// TIA Portal V20 export
FUNCTION_BLOCK "FB_PusherControl"   // FB3, LAD
TITLE = Pusher Control
// Pusher ram sequencing (C-118-C-125). Step legend (C-120): 0=Idle (no motion; home is the HomeLimit switch, not implied by the step - after a jog release the ram may legitimately rest off home, REQ-039) - 10=DriveToEndTravel (forward stroke in progress) - 20=Hold (paused at full travel, brief settle before retracting) - 30=Retract (returning to home; also the recovery/abort target from any bad state). Mode legend: 0=Off (finish a retract already in progress, then park; no new cycle starts) - 1=Auto (hopper-high-level starts a cycle) - 2=Manual (operator button/jog starts a cycle). Motion policy (owner rulings 2026-07-16): an idle off-home ram reparks ONLY on the plant pre-start ParkCmd or on a live cycle request - never on jog release or bare mode changes - and every motion start from rest (repark, cycle launch, jog) is preceded by the JogWarningTime sounder warning (NEW-4: no unwarned pusher motion). CycleInhibit (any live plant stop reason) blocks cycle launches and aborts an in-flight cycle to park, but deliberately leaves hand-jog available - only the mode-0 force (stop button/unhealthy) blocks jogging (owner amendment 2026-07-16, REQ-040). Fitted=FALSE (REQ-042/043/044) kills every demand, the pack output, both supervision timers, and every fault latch at the source, so a disabled pusher does nothing and raises nothing. A live drop mid-cycle also force-parks Step to 0/Idle rather than stranding it non-zero (owner ruling 2026-07-17, B-4, NETWORK 14) - re-enabling Fitted is never itself a start condition (C-128): the normal Step 0 launch/repark gates (NETWORK 1) still require a fresh live trigger before anything moves again.
   VAR RETAIN
      IO { S7_SetPoint := 'True'} : "UDT_PusherIO";   // Caller-visible interface (C-115) - FC_ControlMain writes Mode/HopperHighLevel/limits/tunables in, reads Extend/Retract/RunPowerPack/fault bits out. See the block header for the Step/Mode value legend.
   END_VAR
   VAR
      CycleRequest : Bool;   // Named once, read everywhere (C-601): the live cycle trigger - Auto on hopper high or Manual on the HMI button - gated by Enable (Fitted AND not Off) and NOT Blocked. Read by the warning armer, the launch and repark transitions, and the trip-count reset. Blocked is written later in the scan, so this reads it one scan behind - immaterial: Blocked can only latch mid-stroke (Step 10) where no Step 0 request can act, and a reset-clear merely delays a relaunch by one scan.
      JogDemand : Bool;   // A live jog request: either jog button held, idle, Manual mode, pusher fitted. Arms the pre-motion warning, suppresses the repark (jogging is never fought by an auto-retract), and - per direction, warning done - drives the demands. Reads Step from before this scan's transitions; the demand rungs re-check Step fresh.
      ReparkRequest : Bool;   // A repark to home is wanted: the sequencer's pre-start ParkCmd (REQ-045) or a live CycleRequest, while idle off home and not jogging. One of the only two motion sources out of Step 0 (owner ruling 2026-07-16); fires the 0-to-30 transition once the pre-motion warning has sounded.
      LaunchRequest : Bool;   // A cycle launch is possible: live CycleRequest, idle, ram at home. Fires the 0-to-10 transition once the pre-motion warning has sounded; the same fired condition resets PressureTripCount (per-cycle jam counting, REQ-048).
      CycleAbort : Bool;   // Named once (C-601): abort an in-flight cycle to Retract - Off commanded mid-cycle, or the plant acquired a stop reason (CycleInhibit). Read by the Step 10 and Step 20 exits; the Step 30 retract completes regardless, so an aborted cycle always ends parked. Jog is untouched by this bit (owner amendment 2026-07-16).
      EndTravelTimeoutMS : DInt;
      ParkedTimeoutMS : DInt;
      EndTravelHoldTimeMS : DInt;
      PumpRunOnTimeMS : DInt;
      JogWarningTimeMS : DInt;
      PressureTripConfirmTimeMS : DInt;
      PressureClearResumeDelayMS : DInt;
      PressureConfirmTimer { S7_SetPoint := 'True'} : TON_TIME;
      PressureClearTimer { S7_SetPoint := 'True'} : TON_TIME;
      PressureHold : Bool;   // Latched jam hold, not a fault (C-123) - see the Pressure Detection network. Freezes ExtendDemand while set; clears itself once pressure has genuinely stayed clear for PressureClearResumeDelay.
      PressureConfirmEdge : Bool;
      PressureConfirmEdgeMem : Bool;
      PressureTripCount : Int;   // Confirmed jams this cycle - reset each cycle start, not time-windowed. Compared against IO.PressureTripCountThreshold to raise Blocked.
      EndTravelTimer { S7_SetPoint := 'True'} : TON_TIME;
      HoldTimer { S7_SetPoint := 'True'} : TON_TIME;
      ParkedTimer { S7_SetPoint := 'True'} : TON_TIME;
      JogPreStartTimer { S7_SetPoint := 'True'} : TON_TIME;
      ExtendDemand : Bool;
      RetractDemand : Bool;
      PumpDemand : Bool;   // ExtendDemand OR RetractDemand - the pump's own immediate (non-run-on) demand signal.
      PumpEverDemanded : Bool;   // Cold-start guard for the pump run-on off-delay below - see that network's own comment.
      PumpRunOnTimer { S7_SetPoint := 'True'} : TON_TIME;
   END_VAR
   VAR_TEMP
      "Time" : Real;
   END_VAR
BEGIN

REGION Network 1: Enable And Motion Requests
   // The compound conditions every later network shares, each written once (C-601). Requests read Step as it settled last scan (the transitions run later) - safe, because Step only ever leaves 0 through this scan's own request-gated transitions; steps returning to 0 just re-arm the requests one scan late. CycleInhibit kills cycle requests (no launch into a stopped plant) and, via CycleAbort, retracts an in-flight cycle - while JogDemand deliberately ignores it: hand-jog stays available with the plant stopped by downstream absence (owner amendment 2026-07-16, REQ-040).
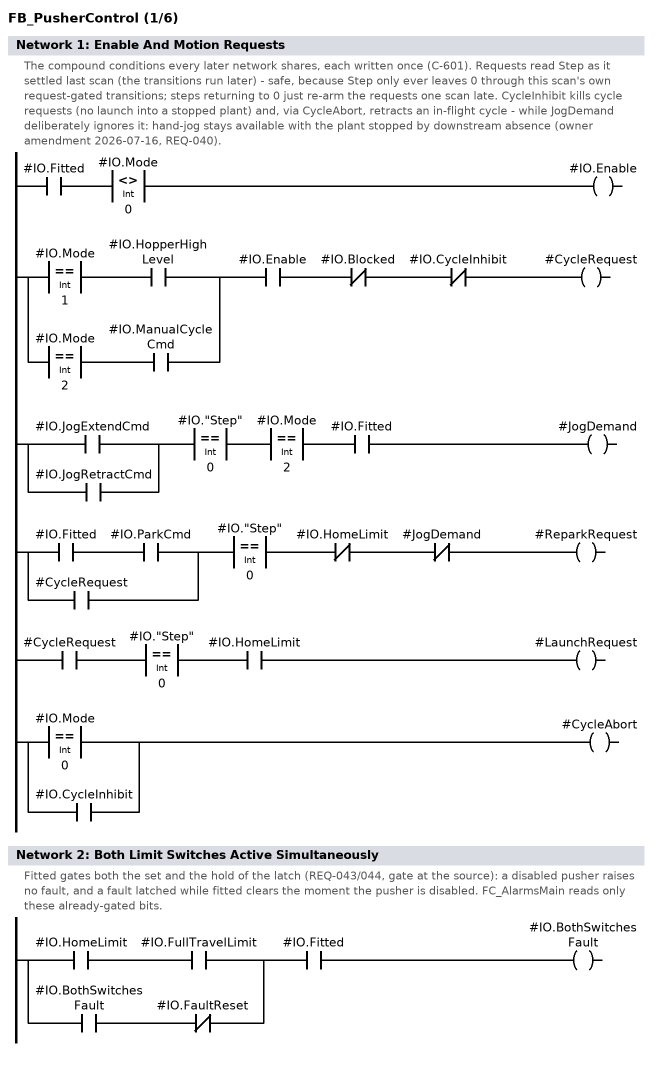
   RUNG wire#powerrail
      Contact( #IO.Fitted )
      { S7_Templates := "SrcType := Int" } NE_Contact(in1 := #IO.Mode, in2 := 0)
      Coil( #IO.Enable )
   END_RUNG
   RUNG wire#powerrail
      { S7_Templates := "SrcType := Int" } EQ_Contact(in1 := #IO.Mode, in2 := 1)
      Contact( #IO.HopperHighLevel )
      wire#w1
      Contact( #IO.Enable )
      I_Contact( #IO.Blocked )
      I_Contact( #IO.CycleInhibit )
      Coil( #CycleRequest )
   END_RUNG
   RUNG wire#powerrail
      { S7_Templates := "SrcType := Int" } EQ_Contact(in1 := #IO.Mode, in2 := 2)
      Contact( #IO.ManualCycleCmd )
   END_RUNG wire#w1
   RUNG wire#powerrail
      Contact( #IO.JogExtendCmd )
      wire#w2
      { S7_Templates := "SrcType := Int" } EQ_Contact(in1 := #IO."Step", in2 := 0)
      { S7_Templates := "SrcType := Int" } EQ_Contact(in1 := #IO.Mode, in2 := 2)
      Contact( #IO.Fitted )
      Coil( #JogDemand )
   END_RUNG
   RUNG wire#powerrail
      Contact( #IO.JogRetractCmd )
   END_RUNG wire#w2
   RUNG wire#powerrail
      Contact( #IO.Fitted )
      Contact( #IO.ParkCmd )
      wire#w3
      { S7_Templates := "SrcType := Int" } EQ_Contact(in1 := #IO."Step", in2 := 0)
      I_Contact( #IO.HomeLimit )
      I_Contact( #JogDemand )
      Coil( #ReparkRequest )
   END_RUNG
   RUNG wire#powerrail
      Contact( #CycleRequest )
   END_RUNG wire#w3
   RUNG wire#powerrail
      Contact( #CycleRequest )
      { S7_Templates := "SrcType := Int" } EQ_Contact(in1 := #IO."Step", in2 := 0)
      Contact( #IO.HomeLimit )
      Coil( #LaunchRequest )
   END_RUNG
   RUNG wire#powerrail
      { S7_Templates := "SrcType := Int" } EQ_Contact(in1 := #IO.Mode, in2 := 0)
      wire#w4
      Coil( #CycleAbort )
   END_RUNG
   RUNG wire#powerrail
      Contact( #IO.CycleInhibit )
   END_RUNG wire#w4
   // the same network as SCL:
   #IO.Enable := #IO.Fitted AND (#IO.Mode <> 0);
   #CycleRequest := (((#IO.Mode = 1) AND #IO.HopperHighLevel) OR ((#IO.Mode = 2) AND #IO.ManualCycleCmd)) AND #IO.Enable AND NOT #IO.Blocked AND NOT #IO.CycleInhibit;
   #JogDemand := (#IO.JogExtendCmd OR #IO.JogRetractCmd) AND (#IO."Step" = 0) AND (#IO.Mode = 2) AND #IO.Fitted;
   #ReparkRequest := ((#IO.Fitted AND #IO.ParkCmd) OR #CycleRequest) AND (#IO."Step" = 0) AND NOT #IO.HomeLimit AND NOT #JogDemand;
   #LaunchRequest := #CycleRequest AND (#IO."Step" = 0) AND #IO.HomeLimit;
   #CycleAbort := (#IO.Mode = 0) OR #IO.CycleInhibit;
END_REGION

REGION Network 2: Both Limit Switches Active Simultaneously
   // Fitted gates both the set and the hold of the latch (REQ-043/044, gate at the source): a disabled pusher raises no fault, and a fault latched while fitted clears the moment the pusher is disabled. FC_AlarmsMain reads only these already-gated bits.
   RUNG wire#powerrail
      Contact( #IO.HomeLimit )
      Contact( #IO.FullTravelLimit )
      wire#w1
      Contact( #IO.Fitted )
      Coil( #IO.BothSwitchesFault )
   END_RUNG
   RUNG wire#powerrail
      Contact( #IO.BothSwitchesFault )
      I_Contact( #IO.FaultReset )
   END_RUNG wire#w1
   // the same network as SCL:
   #IO.BothSwitchesFault := ((#IO.HomeLimit AND #IO.FullTravelLimit) OR (#IO.BothSwitchesFault AND NOT #IO.FaultReset)) AND #IO.Fitted;
END_REGION

REGION Network 3: HMI Time Conversions
   // HMI/DB_Settings times are Real seconds for operator legibility; every TON below needs its PT in DInt ms - one MUL+CONVERT pair per timer, matching the MotorDOL FTTime/EnableUPSTime idiom. Kept as one block up front rather than repeated at each timer, so the x1000 idiom is visibly consistent and only ever done once.
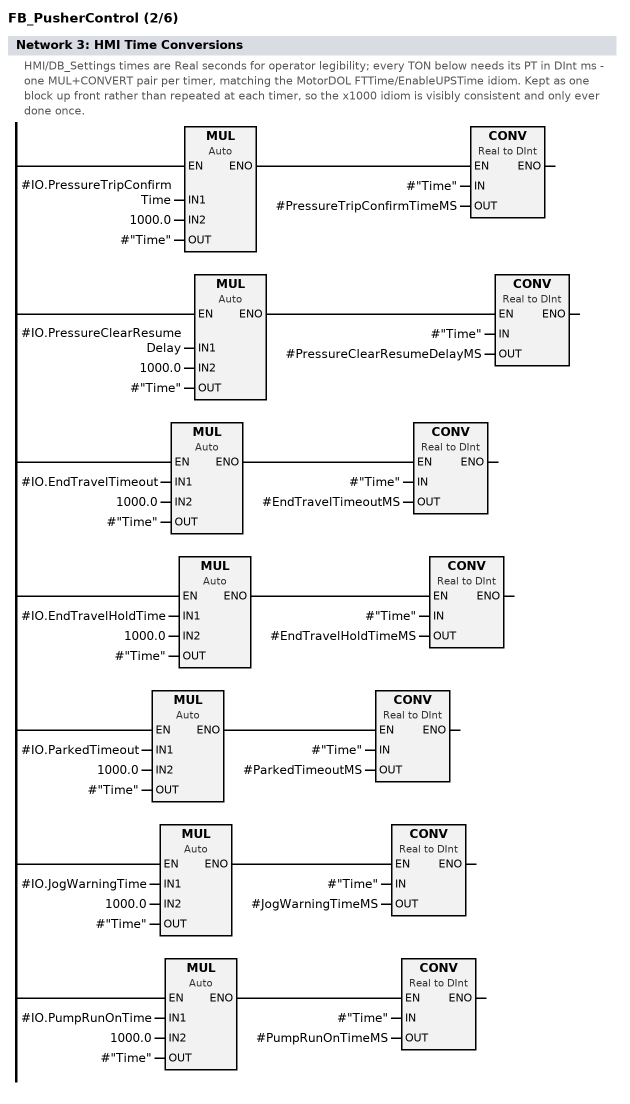
   RUNG wire#powerrail
      Mul(in1 := #IO.PressureTripConfirmTime, in2 := 1000.0, out := #"Time")
      { S7_Templates := "[SrcType := Real, DestType := DInt]" } Convert(in := #"Time", out := #PressureTripConfirmTimeMS)
   END_RUNG
   RUNG wire#powerrail
      Mul(in1 := #IO.PressureClearResumeDelay, in2 := 1000.0, out := #"Time")
      { S7_Templates := "[SrcType := Real, DestType := DInt]" } Convert(in := #"Time", out := #PressureClearResumeDelayMS)
   END_RUNG
   RUNG wire#powerrail
      Mul(in1 := #IO.EndTravelTimeout, in2 := 1000.0, out := #"Time")
      { S7_Templates := "[SrcType := Real, DestType := DInt]" } Convert(in := #"Time", out := #EndTravelTimeoutMS)
   END_RUNG
   RUNG wire#powerrail
      Mul(in1 := #IO.EndTravelHoldTime, in2 := 1000.0, out := #"Time")
      { S7_Templates := "[SrcType := Real, DestType := DInt]" } Convert(in := #"Time", out := #EndTravelHoldTimeMS)
   END_RUNG
   RUNG wire#powerrail
      Mul(in1 := #IO.ParkedTimeout, in2 := 1000.0, out := #"Time")
      { S7_Templates := "[SrcType := Real, DestType := DInt]" } Convert(in := #"Time", out := #ParkedTimeoutMS)
   END_RUNG
   RUNG wire#powerrail
      Mul(in1 := #IO.JogWarningTime, in2 := 1000.0, out := #"Time")
      { S7_Templates := "[SrcType := Real, DestType := DInt]" } Convert(in := #"Time", out := #JogWarningTimeMS)
   END_RUNG
   RUNG wire#powerrail
      Mul(in1 := #IO.PumpRunOnTime, in2 := 1000.0, out := #"Time")
      { S7_Templates := "[SrcType := Real, DestType := DInt]" } Convert(in := #"Time", out := #PumpRunOnTimeMS)
   END_RUNG
   // the same network as SCL:
   <??.?> := #IO.PressureTripConfirmTime * 1000.0 * #"Time";
   <??.?> := REAL_TO_DINT(#"Time");
   <??.?> := #IO.PressureClearResumeDelay * 1000.0 * #"Time";
   <??.?> := REAL_TO_DINT(#"Time");
   <??.?> := #IO.EndTravelTimeout * 1000.0 * #"Time";
   <??.?> := REAL_TO_DINT(#"Time");
   <??.?> := #IO.EndTravelHoldTime * 1000.0 * #"Time";
   <??.?> := REAL_TO_DINT(#"Time");
   <??.?> := #IO.ParkedTimeout * 1000.0 * #"Time";
   <??.?> := REAL_TO_DINT(#"Time");
   <??.?> := #IO.JogWarningTime * 1000.0 * #"Time";
   <??.?> := REAL_TO_DINT(#"Time");
   <??.?> := #IO.PumpRunOnTime * 1000.0 * #"Time";
   <??.?> := REAL_TO_DINT(#"Time");
END_REGION

REGION Network 4: Pre-Motion Warning
   // NEW-4 owner ruling (2026-07-16): no unwarned pusher motion. Every motion start from rest - repark, auto/manual cycle launch, jog - arms this timer and the sounder; the Step 0 transitions and the jog demands only act on its Q, so the sounder always leads motion by JogWarningTime. Jog keeps sounding while moving (REQ-041) because JogDemand stays true through the jog; in-cycle strokes (10/20/30, including a stop-forced retract) are continuations of an already-warned launch, so the warning boundary is Step 0. A request released mid-warning (short manual tap, hopper clearing) simply never moves. Timer and sounder keep their original jog-era names to avoid interface churn - rename queued with the cosmetic pass.
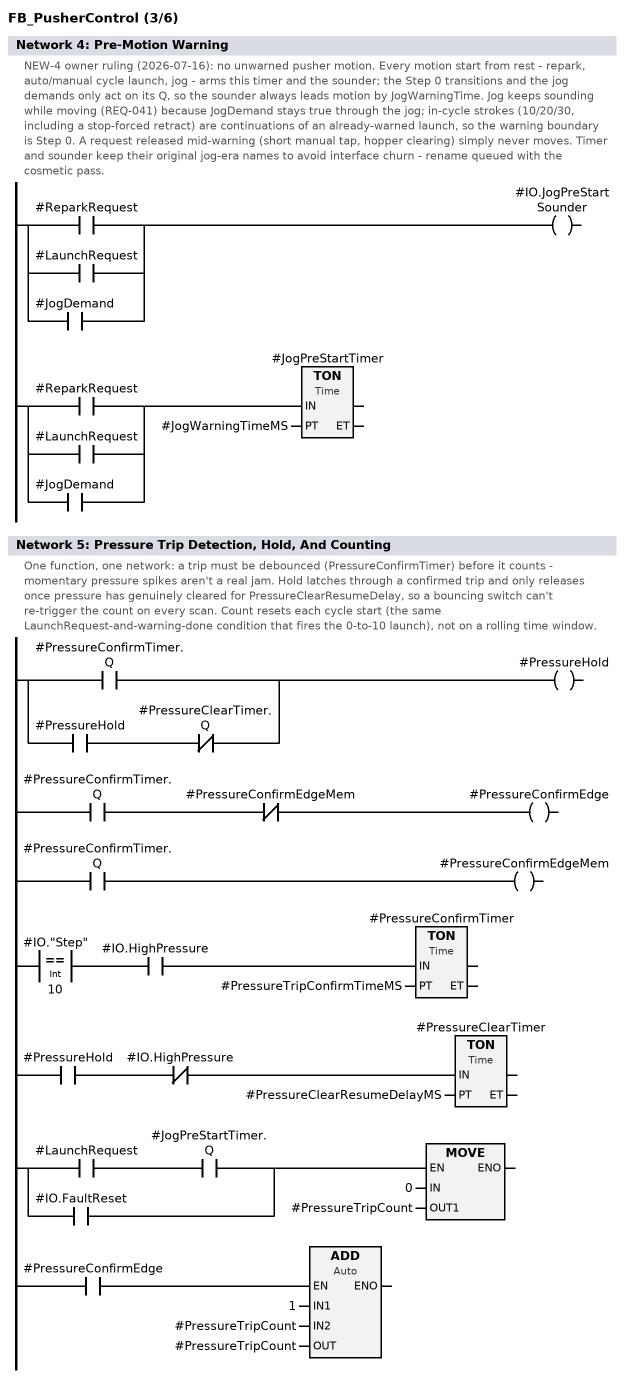
   RUNG wire#powerrail
      Contact( #ReparkRequest )
      wire#w1
      Coil( #IO.JogPreStartSounder )
   END_RUNG
   RUNG wire#powerrail
      Contact( #LaunchRequest )
   END_RUNG wire#w1
   RUNG wire#powerrail
      Contact( #JogDemand )
   END_RUNG wire#w1
   RUNG wire#powerrail
      Contact( #ReparkRequest )
      wire#w2
      { S7_Templates := "time_type := Time" } #JogPreStartTimer.TON(pt := #JogWarningTimeMS, et =>)
   END_RUNG
   RUNG wire#powerrail
      Contact( #LaunchRequest )
   END_RUNG wire#w2
   RUNG wire#powerrail
      Contact( #JogDemand )
   END_RUNG wire#w2
   // the same network as SCL:
   #IO.JogPreStartSounder := #ReparkRequest OR #LaunchRequest OR #JogDemand;
   #JogPreStartTimer(IN := #ReparkRequest OR #LaunchRequest OR #JogDemand, PT := #JogWarningTimeMS);   // TON
END_REGION

REGION Network 5: Pressure Trip Detection, Hold, And Counting
   // One function, one network: a trip must be debounced (PressureConfirmTimer) before it counts - momentary pressure spikes aren't a real jam. Hold latches through a confirmed trip and only releases once pressure has genuinely cleared for PressureClearResumeDelay, so a bouncing switch can't re-trigger the count on every scan. Count resets each cycle start (the same LaunchRequest-and-warning-done condition that fires the 0-to-10 launch), not on a rolling time window.
   RUNG wire#powerrail
      Contact( #PressureConfirmTimer.Q )
      wire#w1
      Coil( #PressureHold )
   END_RUNG
   RUNG wire#powerrail
      Contact( #PressureHold )
      I_Contact( #PressureClearTimer.Q )
   END_RUNG wire#w1
   RUNG wire#powerrail
      Contact( #PressureConfirmTimer.Q )
      I_Contact( #PressureConfirmEdgeMem )
      Coil( #PressureConfirmEdge )
   END_RUNG
   RUNG wire#powerrail
      Contact( #PressureConfirmTimer.Q )
      Coil( #PressureConfirmEdgeMem )
   END_RUNG
   RUNG wire#powerrail
      { S7_Templates := "SrcType := Int" } EQ_Contact(in1 := #IO."Step", in2 := 10)
      Contact( #IO.HighPressure )
      { S7_Templates := "time_type := Time" } #PressureConfirmTimer.TON(pt := #PressureTripConfirmTimeMS, et =>)
   END_RUNG
   RUNG wire#powerrail
      Contact( #PressureHold )
      I_Contact( #IO.HighPressure )
      { S7_Templates := "time_type := Time" } #PressureClearTimer.TON(pt := #PressureClearResumeDelayMS, et =>)
   END_RUNG
   RUNG wire#powerrail
      Contact( #LaunchRequest )
      Contact( #JogPreStartTimer.Q )
      wire#w2
      Move(in := 0, out1 := #PressureTripCount)
   END_RUNG
   RUNG wire#powerrail
      Contact( #IO.FaultReset )
   END_RUNG wire#w2
   RUNG wire#powerrail
      Contact( #PressureConfirmEdge )
      Add(in1 := 1, in2 := #PressureTripCount, out := #PressureTripCount)
   END_RUNG
   // the same network as SCL:
   #PressureHold := #PressureConfirmTimer.Q OR (#PressureHold AND NOT #PressureClearTimer.Q);
   #PressureConfirmEdge := #PressureConfirmTimer.Q AND NOT #PressureConfirmEdgeMem;
   #PressureConfirmEdgeMem := #PressureConfirmTimer.Q;
   #PressureConfirmTimer(IN := (#IO."Step" = 10) AND #IO.HighPressure, PT := #PressureTripConfirmTimeMS);   // TON
   #PressureClearTimer(IN := #PressureHold AND NOT #IO.HighPressure, PT := #PressureClearResumeDelayMS);   // TON
   IF (#LaunchRequest AND #JogPreStartTimer.Q) OR #IO.FaultReset THEN <??.?> := 0; END_IF;
   IF #PressureConfirmEdge THEN <??.?> := 1 + #PressureTripCount + #PressureTripCount; END_IF;
END_REGION

REGION Network 6: Blocked Fault (Too Many Jams)
   // Fitted gates set and hold (REQ-043/044, gate at the source) - a disabled pusher raises nothing, and disabling clears a standing latch.
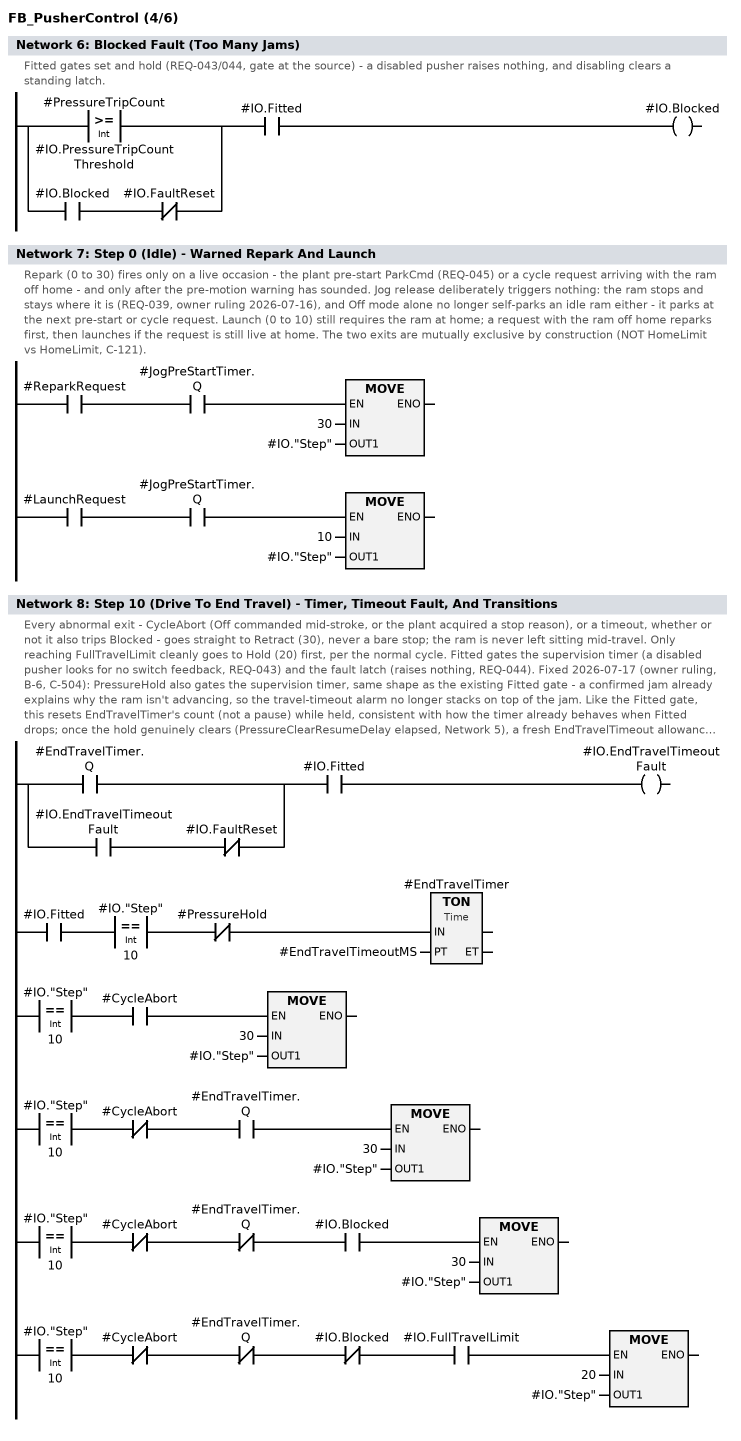
   RUNG wire#powerrail
      { S7_Templates := "SrcType := Int" } GE_Contact(in1 := #PressureTripCount, in2 := #IO.PressureTripCountThreshold)
      wire#w1
      Contact( #IO.Fitted )
      Coil( #IO.Blocked )
   END_RUNG
   RUNG wire#powerrail
      Contact( #IO.Blocked )
      I_Contact( #IO.FaultReset )
   END_RUNG wire#w1
   // the same network as SCL:
   #IO.Blocked := ((#PressureTripCount >= #IO.PressureTripCountThreshold) OR (#IO.Blocked AND NOT #IO.FaultReset)) AND #IO.Fitted;
END_REGION

REGION Network 7: Step 0 (Idle) - Warned Repark And Launch
   // Repark (0 to 30) fires only on a live occasion - the plant pre-start ParkCmd (REQ-045) or a cycle request arriving with the ram off home - and only after the pre-motion warning has sounded. Jog release deliberately triggers nothing: the ram stops and stays where it is (REQ-039, owner ruling 2026-07-16), and Off mode alone no longer self-parks an idle ram either - it parks at the next pre-start or cycle request. Launch (0 to 10) still requires the ram at home; a request with the ram off home reparks first, then launches if the request is still live at home. The two exits are mutually exclusive by construction (NOT HomeLimit vs HomeLimit, C-121).
   RUNG wire#powerrail
      Contact( #ReparkRequest )
      Contact( #JogPreStartTimer.Q )
      Move(in := 30, out1 := #IO."Step")
   END_RUNG
   RUNG wire#powerrail
      Contact( #LaunchRequest )
      Contact( #JogPreStartTimer.Q )
      Move(in := 10, out1 := #IO."Step")
   END_RUNG
   // the same network as SCL:
   IF #ReparkRequest AND #JogPreStartTimer.Q THEN <??.?> := 30; END_IF;
   IF #LaunchRequest AND #JogPreStartTimer.Q THEN <??.?> := 10; END_IF;
END_REGION

REGION Network 8: Step 10 (Drive To End Travel) - Timer, Timeout Fault, And Transitions
   // Every abnormal exit - CycleAbort (Off commanded mid-stroke, or the plant acquired a stop reason), or a timeout, whether or not it also trips Blocked - goes straight to Retract (30), never a bare stop; the ram is never left sitting mid-travel. Only reaching FullTravelLimit cleanly goes to Hold (20) first, per the normal cycle. Fitted gates the supervision timer (a disabled pusher looks for no switch feedback, REQ-043) and the fault latch (raises nothing, REQ-044). Fixed 2026-07-17 (owner ruling, B-6, C-504): PressureHold also gates the supervision timer, same shape as the existing Fitted gate - a confirmed jam already explains why the ram isn't advancing, so the travel-timeout alarm no longer stacks on top of the jam. Like the Fitted gate, this resets EndTravelTimer's count (not a pause) while held, consistent with how the timer already behaves when Fitted drops; once the hold genuinely clears (PressureClearResumeDelay elapsed, Network 5), a fresh EndTravelTimeout allowance starts - if the ram still doesn't reach FullTravelLimit within that, the timeout is real, not an echo of the jam.
   RUNG wire#powerrail
      Contact( #EndTravelTimer.Q )
      wire#w1
      Contact( #IO.Fitted )
      Coil( #IO.EndTravelTimeoutFault )
   END_RUNG
   RUNG wire#powerrail
      Contact( #IO.EndTravelTimeoutFault )
      I_Contact( #IO.FaultReset )
   END_RUNG wire#w1
   RUNG wire#powerrail
      Contact( #IO.Fitted )
      { S7_Templates := "SrcType := Int" } EQ_Contact(in1 := #IO."Step", in2 := 10)
      I_Contact( #PressureHold )
      { S7_Templates := "time_type := Time" } #EndTravelTimer.TON(pt := #EndTravelTimeoutMS, et =>)
   END_RUNG
   RUNG wire#powerrail
      { S7_Templates := "SrcType := Int" } EQ_Contact(in1 := #IO."Step", in2 := 10)
      Contact( #CycleAbort )
      Move(in := 30, out1 := #IO."Step")
   END_RUNG
   RUNG wire#powerrail
      { S7_Templates := "SrcType := Int" } EQ_Contact(in1 := #IO."Step", in2 := 10)
      I_Contact( #CycleAbort )
      Contact( #EndTravelTimer.Q )
      Move(in := 30, out1 := #IO."Step")
   END_RUNG
   RUNG wire#powerrail
      { S7_Templates := "SrcType := Int" } EQ_Contact(in1 := #IO."Step", in2 := 10)
      I_Contact( #CycleAbort )
      I_Contact( #EndTravelTimer.Q )
      Contact( #IO.Blocked )
      Move(in := 30, out1 := #IO."Step")
   END_RUNG
   RUNG wire#powerrail
      { S7_Templates := "SrcType := Int" } EQ_Contact(in1 := #IO."Step", in2 := 10)
      I_Contact( #CycleAbort )
      I_Contact( #EndTravelTimer.Q )
      I_Contact( #IO.Blocked )
      Contact( #IO.FullTravelLimit )
      Move(in := 20, out1 := #IO."Step")
   END_RUNG
   // the same network as SCL:
   #IO.EndTravelTimeoutFault := (#EndTravelTimer.Q OR (#IO.EndTravelTimeoutFault AND NOT #IO.FaultReset)) AND #IO.Fitted;
   #EndTravelTimer(IN := #IO.Fitted AND (#IO."Step" = 10) AND NOT #PressureHold, PT := #EndTravelTimeoutMS);   // TON
   IF (#IO."Step" = 10) AND #CycleAbort THEN <??.?> := 30; END_IF;
   IF (#IO."Step" = 10) AND NOT #CycleAbort AND #EndTravelTimer.Q THEN <??.?> := 30; END_IF;
   IF (#IO."Step" = 10) AND NOT #CycleAbort AND NOT #EndTravelTimer.Q AND #IO.Blocked THEN
       <??.?> := 30;
   END_IF;
   IF (#IO."Step" = 10) AND NOT #CycleAbort AND NOT #EndTravelTimer.Q AND NOT #IO.Blocked AND #IO.FullTravelLimit THEN
       <??.?> := 20;
   END_IF;
END_REGION

REGION Network 9: Step 20 (Hold) - Timer And Transition
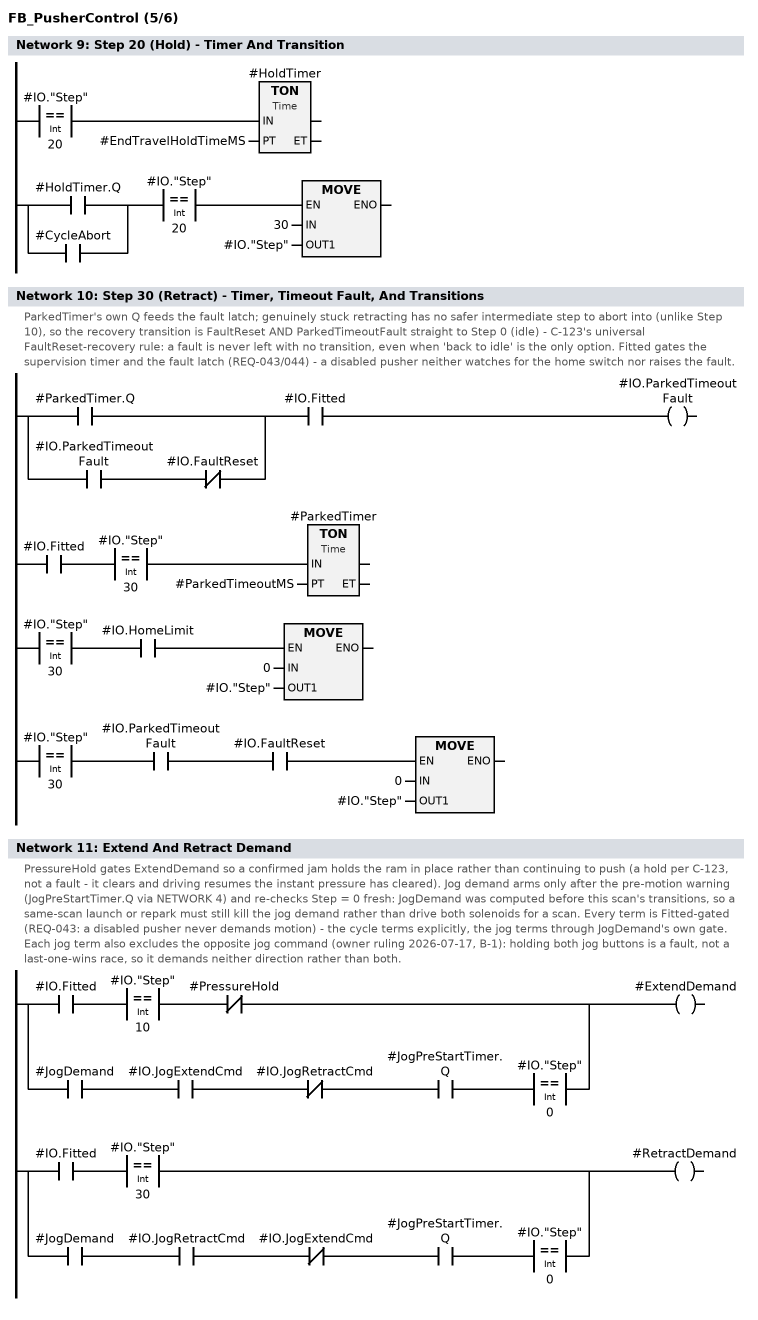
   RUNG wire#powerrail
      { S7_Templates := "SrcType := Int" } EQ_Contact(in1 := #IO."Step", in2 := 20)
      { S7_Templates := "time_type := Time" } #HoldTimer.TON(pt := #EndTravelHoldTimeMS, et =>)
   END_RUNG
   RUNG wire#powerrail
      Contact( #HoldTimer.Q )
      wire#w1
      { S7_Templates := "SrcType := Int" } EQ_Contact(in1 := #IO."Step", in2 := 20)
      Move(in := 30, out1 := #IO."Step")
   END_RUNG
   RUNG wire#powerrail
      Contact( #CycleAbort )
   END_RUNG wire#w1
   // the same network as SCL:
   #HoldTimer(IN := #IO."Step" = 20, PT := #EndTravelHoldTimeMS);   // TON
   IF (#HoldTimer.Q OR #CycleAbort) AND (#IO."Step" = 20) THEN <??.?> := 30; END_IF;
END_REGION

REGION Network 10: Step 30 (Retract) - Timer, Timeout Fault, And Transitions
   // ParkedTimer's own Q feeds the fault latch; genuinely stuck retracting has no safer intermediate step to abort into (unlike Step 10), so the recovery transition is FaultReset AND ParkedTimeoutFault straight to Step 0 (idle) - C-123's universal FaultReset-recovery rule: a fault is never left with no transition, even when 'back to idle' is the only option. Fitted gates the supervision timer and the fault latch (REQ-043/044) - a disabled pusher neither watches for the home switch nor raises the fault.
   RUNG wire#powerrail
      Contact( #ParkedTimer.Q )
      wire#w1
      Contact( #IO.Fitted )
      Coil( #IO.ParkedTimeoutFault )
   END_RUNG
   RUNG wire#powerrail
      Contact( #IO.ParkedTimeoutFault )
      I_Contact( #IO.FaultReset )
   END_RUNG wire#w1
   RUNG wire#powerrail
      Contact( #IO.Fitted )
      { S7_Templates := "SrcType := Int" } EQ_Contact(in1 := #IO."Step", in2 := 30)
      { S7_Templates := "time_type := Time" } #ParkedTimer.TON(pt := #ParkedTimeoutMS, et =>)
   END_RUNG
   RUNG wire#powerrail
      { S7_Templates := "SrcType := Int" } EQ_Contact(in1 := #IO."Step", in2 := 30)
      Contact( #IO.HomeLimit )
      Move(in := 0, out1 := #IO."Step")
   END_RUNG
   RUNG wire#powerrail
      { S7_Templates := "SrcType := Int" } EQ_Contact(in1 := #IO."Step", in2 := 30)
      Contact( #IO.ParkedTimeoutFault )
      Contact( #IO.FaultReset )
      Move(in := 0, out1 := #IO."Step")
   END_RUNG
   // the same network as SCL:
   #IO.ParkedTimeoutFault := (#ParkedTimer.Q OR (#IO.ParkedTimeoutFault AND NOT #IO.FaultReset)) AND #IO.Fitted;
   #ParkedTimer(IN := #IO.Fitted AND (#IO."Step" = 30), PT := #ParkedTimeoutMS);   // TON
   IF (#IO."Step" = 30) AND #IO.HomeLimit THEN <??.?> := 0; END_IF;
   IF (#IO."Step" = 30) AND #IO.ParkedTimeoutFault AND #IO.FaultReset THEN <??.?> := 0; END_IF;
END_REGION

REGION Network 11: Extend And Retract Demand
   // PressureHold gates ExtendDemand so a confirmed jam holds the ram in place rather than continuing to push (a hold per C-123, not a fault - it clears and driving resumes the instant pressure has cleared). Jog demand arms only after the pre-motion warning (JogPreStartTimer.Q via NETWORK 4) and re-checks Step = 0 fresh: JogDemand was computed before this scan's transitions, so a same-scan launch or repark must still kill the jog demand rather than drive both solenoids for a scan. Every term is Fitted-gated (REQ-043: a disabled pusher never demands motion) - the cycle terms explicitly, the jog terms through JogDemand's own gate. Each jog term also excludes the opposite jog command (owner ruling 2026-07-17, B-1): holding both jog buttons is a fault, not a last-one-wins race, so it demands neither direction rather than both.
   RUNG wire#powerrail
      Contact( #IO.Fitted )
      { S7_Templates := "SrcType := Int" } EQ_Contact(in1 := #IO."Step", in2 := 10)
      I_Contact( #PressureHold )
      wire#w1
      Coil( #ExtendDemand )
   END_RUNG
   RUNG wire#powerrail
      Contact( #JogDemand )
      Contact( #IO.JogExtendCmd )
      I_Contact( #IO.JogRetractCmd )
      Contact( #JogPreStartTimer.Q )
      { S7_Templates := "SrcType := Int" } EQ_Contact(in1 := #IO."Step", in2 := 0)
   END_RUNG wire#w1
   RUNG wire#powerrail
      Contact( #IO.Fitted )
      { S7_Templates := "SrcType := Int" } EQ_Contact(in1 := #IO."Step", in2 := 30)
      wire#w2
      Coil( #RetractDemand )
   END_RUNG
   RUNG wire#powerrail
      Contact( #JogDemand )
      Contact( #IO.JogRetractCmd )
      I_Contact( #IO.JogExtendCmd )
      Contact( #JogPreStartTimer.Q )
      { S7_Templates := "SrcType := Int" } EQ_Contact(in1 := #IO."Step", in2 := 0)
   END_RUNG wire#w2
   // the same network as SCL:
   #ExtendDemand := (#IO.Fitted AND (#IO."Step" = 10) AND NOT #PressureHold) OR (#JogDemand AND #IO.JogExtendCmd AND NOT #IO.JogRetractCmd AND #JogPreStartTimer.Q AND (#IO."Step" = 0));
   #RetractDemand := (#IO.Fitted AND (#IO."Step" = 30)) OR (#JogDemand AND #IO.JogRetractCmd AND NOT #IO.JogExtendCmd AND #JogPreStartTimer.Q AND (#IO."Step" = 0));
END_REGION

REGION Network 12: Pump Demand
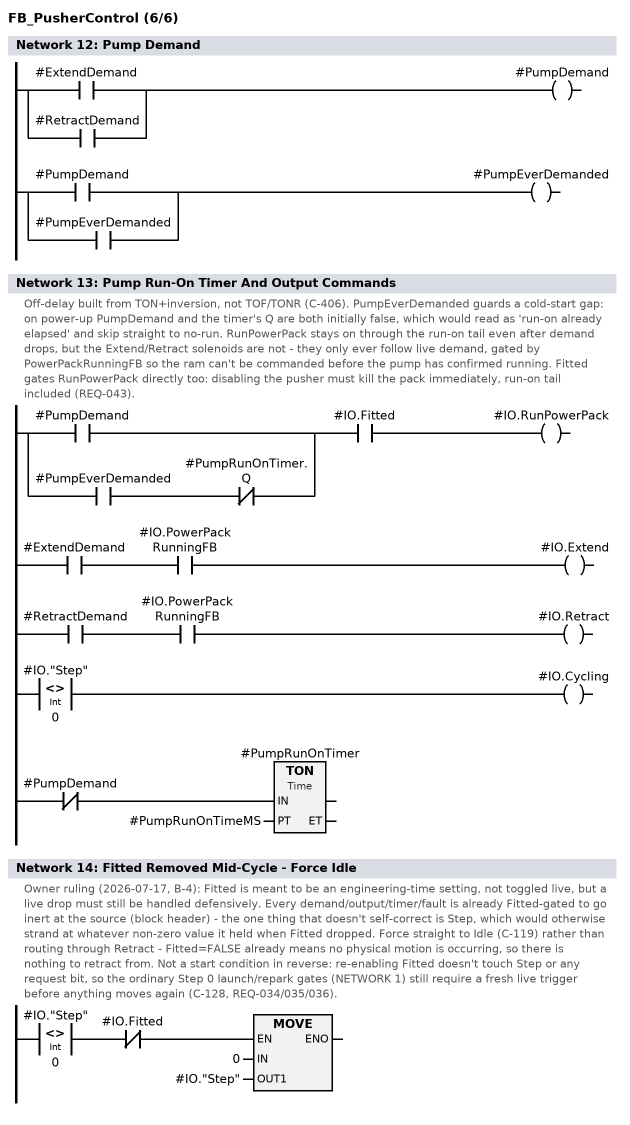
   RUNG wire#powerrail
      Contact( #ExtendDemand )
      wire#w1
      Coil( #PumpDemand )
   END_RUNG
   RUNG wire#powerrail
      Contact( #RetractDemand )
   END_RUNG wire#w1
   RUNG wire#powerrail
      Contact( #PumpDemand )
      wire#w2
      Coil( #PumpEverDemanded )
   END_RUNG
   RUNG wire#powerrail
      Contact( #PumpEverDemanded )
   END_RUNG wire#w2
   // the same network as SCL:
   #PumpDemand := #ExtendDemand OR #RetractDemand;
   #PumpEverDemanded := #PumpDemand OR #PumpEverDemanded;
END_REGION

REGION Network 13: Pump Run-On Timer And Output Commands
   // Off-delay built from TON+inversion, not TOF/TONR (C-406). PumpEverDemanded guards a cold-start gap: on power-up PumpDemand and the timer's Q are both initially false, which would read as 'run-on already elapsed' and skip straight to no-run. RunPowerPack stays on through the run-on tail even after demand drops, but the Extend/Retract solenoids are not - they only ever follow live demand, gated by PowerPackRunningFB so the ram can't be commanded before the pump has confirmed running. Fitted gates RunPowerPack directly too: disabling the pusher must kill the pack immediately, run-on tail included (REQ-043).
   RUNG wire#powerrail
      Contact( #PumpDemand )
      wire#w1
      Contact( #IO.Fitted )
      Coil( #IO.RunPowerPack )
   END_RUNG
   RUNG wire#powerrail
      Contact( #PumpEverDemanded )
      I_Contact( #PumpRunOnTimer.Q )
   END_RUNG wire#w1
   RUNG wire#powerrail
      Contact( #ExtendDemand )
      Contact( #IO.PowerPackRunningFB )
      Coil( #IO.Extend )
   END_RUNG
   RUNG wire#powerrail
      Contact( #RetractDemand )
      Contact( #IO.PowerPackRunningFB )
      Coil( #IO.Retract )
   END_RUNG
   RUNG wire#powerrail
      { S7_Templates := "SrcType := Int" } NE_Contact(in1 := #IO."Step", in2 := 0)
      Coil( #IO.Cycling )
   END_RUNG
   RUNG wire#powerrail
      I_Contact( #PumpDemand )
      { S7_Templates := "time_type := Time" } #PumpRunOnTimer.TON(pt := #PumpRunOnTimeMS, et =>)
   END_RUNG
   // the same network as SCL:
   #IO.RunPowerPack := (#PumpDemand OR (#PumpEverDemanded AND NOT #PumpRunOnTimer.Q)) AND #IO.Fitted;
   #IO.Extend := #ExtendDemand AND #IO.PowerPackRunningFB;
   #IO.Retract := #RetractDemand AND #IO.PowerPackRunningFB;
   #IO.Cycling := #IO."Step" <> 0;
   #PumpRunOnTimer(IN := NOT #PumpDemand, PT := #PumpRunOnTimeMS);   // TON
END_REGION

REGION Network 14: Fitted Removed Mid-Cycle - Force Idle
   // Owner ruling (2026-07-17, B-4): Fitted is meant to be an engineering-time setting, not toggled live, but a live drop must still be handled defensively. Every demand/output/timer/fault is already Fitted-gated to go inert at the source (block header) - the one thing that doesn't self-correct is Step, which would otherwise strand at whatever non-zero value it held when Fitted dropped. Force straight to Idle (C-119) rather than routing through Retract - Fitted=FALSE already means no physical motion is occurring, so there is nothing to retract from. Not a start condition in reverse: re-enabling Fitted doesn't touch Step or any request bit, so the ordinary Step 0 launch/repark gates (NETWORK 1) still require a fresh live trigger before anything moves again (C-128, REQ-034/035/036).
   RUNG wire#powerrail
      { S7_Templates := "SrcType := Int" } NE_Contact(in1 := #IO."Step", in2 := 0)
      I_Contact( #IO.Fitted )
      Move(in := 0, out1 := #IO."Step")
   END_RUNG
   // the same network as SCL:
   IF (#IO."Step" <> 0) AND NOT #IO.Fitted THEN <??.?> := 0; END_IF;
END_REGION
END_FUNCTION_BLOCK
